{attribute 'linkalways'} 
{attribute 'no_explicit_call' := 'This FB is a CLASS and must be accessed using methods or properties'}
{attribute 'enable_dynamic_creation'}
FUNCTION_BLOCK _UDINT EXTENDS NumericDatatypeBase
VAR
	localData : UDINT;
	activeData : REFERENCE TO UDINT REF= localData;
END_VAR

PROPERTY PUBLIC Address : PVOID
GET
Address := ADR(activeData);
END_GET
END_PROPERTY

METHOD PUBLIC ClearReference
VAR_INPUT
END_VAR
activeData REF= localData;
END_METHOD

METHOD PUBLIC Clone : I_Datatype
VAR
    pClone : POINTER TO _UDINT;
END_VAR
pClone := __NEW(_UDINT(InitialValue := Value));
Clone := pClone^;
END_METHOD

METHOD FB_init : BOOL
VAR_INPUT
	bInitRetains : BOOL; // if TRUE, the retain variables are initialized (warm start / cold start)
	bInCopyCode : BOOL;  // if TRUE, the instance afterwards gets moved into the copy code (online change)
	InitialValue : UDINT;
END_VAR
localData := InitialValue;
END_METHOD

PROPERTY PUBLIC IsFloat : BOOL
GET
IsFloat := FALSE;
END_GET
END_PROPERTY

PROPERTY PUBLIC IsSigned : BOOL
GET
IsSigned := FALSE;
END_GET
END_PROPERTY

METHOD PUBLIC MakeReferenceTo
VAR_INPUT
	ReferenceTarget : REFERENCE TO UDINT;
END_VAR
activeData REF= ReferenceTarget;
END_METHOD

PROPERTY PUBLIC MaxValue : UDINT
GET
MaxValue :=  DatatypeLimits.UDINT_MAX_VALUE;
END_GET
END_PROPERTY

PROPERTY PUBLIC MinValue : UDINT
GET
MinValue := DatatypeLimits.UDINT_MIN_VALUE;
END_GET
END_PROPERTY

METHOD PROTECTED SerializeMaxValue
VAR_INPUT
	Serializer : I_Serializer;
END_VAR
Serializer.AddUdint(MaxValue);
END_METHOD

METHOD PROTECTED SerializeMinValue
VAR_INPUT
	Serializer : I_Serializer;
END_VAR
Serializer.AddUdint(MinValue);
END_METHOD

METHOD PUBLIC SerializeWith
VAR_INPUT
	Serializer : I_Serializer;
END_VAR
Serializer.AddUdint(activeData);
END_METHOD

PROPERTY PUBLIC Size : UDINT
GET
Size := SIZEOF(activeData);
END_GET
END_PROPERTY

METHOD TryDeserializeFrom : BOOL
VAR_INPUT
	Deserializer : I_Deserializer;
	Feedback : I_DeserializerFeedback;
END_VAR
TryDeserializeFrom := Deserializer.TryGetUdint(activeData, Feedback);
END_METHOD

METHOD TryMakeReferenceTo : BOOL
VAR_INPUT
	Target : I_Datatype;
END_VAR
VAR
	pTargetData : POINTER TO UDINT;
END_VAR
IF NOT (Target.TypeName = TypeName) THEN
	RETURN;
END_IF

pTargetData := Target.Address;
activeData REF= pTargetData^;
TryMakeReferenceTo := TRUE;
END_METHOD

PROPERTY PUBLIC TypeName : T_MAXSTRING
GET
TypeName := 'UDINT';
END_GET
END_PROPERTY

PROPERTY PUBLIC Value : UDINT
GET
Value := activeData;
END_GET
SET
activeData := Value;
END_SET
END_PROPERTY

END_FUNCTION_BLOCK

(* stored: Version 1.1.0.1, ProductVersion 3.1.4024.12
   POU _UDINT: Id {9b5b5dee-ece4-4773-927d-82d406ffff9a}, SpecialFunc None
   Folder Constructor: Id {5294e336-24fc-4748-b8c5-4a079520937d}
   Folder Protected: Id {9828943b-ecdb-4df8-89a6-013b711dddcd}
   Property Address: Id {81a7983e-63e4-4337-95c8-cc8d9fd48984}
   Get Get: Id {dbf77340-dafd-4c29-953b-9e9261eb0f5e}
   Method ClearReference: Id {ffb809d0-2f98-4348-8031-b8fc8111e19e}
   Method Clone: Id {a5ccc407-fc56-4110-8b1b-a1f5845b47dc}
   Method FB_init: Id {f8c7dd55-cae1-4d36-87c7-69ffd49d8854}
   Property IsFloat: Id {6a90e46c-fabd-4b3e-9388-428ac59f0b01}
   Get Get: Id {d085b73a-8259-4a8f-9e7f-bf585c255ed3}
   Property IsSigned: Id {826feff4-dcbd-4524-bc33-ef0ae2edd56e}
   Get Get: Id {cddf6a78-6b46-42aa-a4df-fbfa32ace517}
   Method MakeReferenceTo: Id {9645a894-a284-4c59-aa37-51d78fe1d883}
   Property MaxValue: Id {5f7279a4-6f3f-4b18-aa02-6a2395494a97}
   Get Get: Id {7e9ebad8-6779-4ddf-9078-2cbdd3a37682}
   Property MinValue: Id {8060f1f0-ec09-4bd2-bfb5-fe891d77bf85}
   Get Get: Id {b9f8b607-c390-48aa-b4c0-a60ce927e079}
   Method SerializeMaxValue: Id {6b3b7fe7-7c5e-4243-9c94-0133beb9582f}
   Method SerializeMinValue: Id {9eefe6a2-8117-4187-9192-a4203345114f}
   Method SerializeWith: Id {21451b5d-0e1c-47b4-a25e-9d56762c703c}
   Property Size: Id {033337ce-8721-44a0-a4f1-2192c8b366a8}
   Get Get: Id {12fbeb4f-90dc-47a5-968a-151f881e90b9}
   Method TryDeserializeFrom: Id {fd0c5ef5-092a-4b41-ad5e-ebdd0d8b48d4}
   Method TryMakeReferenceTo: Id {93edcb17-c259-43de-bbd1-c9ada0bd198e}
   Property TypeName: Id {da8d35b2-9660-4a5d-8a8a-21fb8078915f}
   Get Get: Id {2c7f23a9-0e0b-410b-87ee-5cdddd684529}
   Property Value: Id {5165a7a9-f1f7-4432-ad84-8f184784b43c}
   Get Get: Id {f1af6b3d-7db1-4fd8-aeb7-5b2eba36966d}
   Set Set: Id {c1b8d7b2-8e93-410f-9164-bbac055a0f82} *)
